{attribute 'qualified_only'}
VAR_GLOBAL
	input1 : INT;
END_VAR

(* stored: Version 1.1.0.1, ProductVersion 3.1.4024.9
   GVL GVL_IO: Id {66e3d1e2-2bf1-4049-a9c9-976978cd47df} *)
